(* PLC project Generated.project, CODESYS CODESYS V3.5 SP19 Patch 1 *)
(* stored: creationDateTime 2026-07-27T13:56:34.388274, modificationDateTime 2026-07-27T13:56:34.388274 *)

TYPE ST_Chain_Winch_Demandes : STRUCT
  Idx201_JoyRawPhysical_ANA : INT;  (* [pts] Bruts convertisseur (-2048 à +2048) *)
  Idx202_JoyScaledPhysical_Pct : REAL;  (* [%] Consigne Joystick (-100% à +100%) *)
  Idx203_HmiManualCmd_BtnUp : BOOL;  (* 1 = Appui Bouton Montée IHM | 0 = Relâché *)
  Idx204_HmiManualCmd_BtnDown : BOOL;  (* 1 = Appui Bouton Descente IHM | 0 = Relâché *)
  Idx205_CycleAutoCmd_Pct : REAL;  (* [%] Consigne auto envoyée par le Cycle *)
  Idx206_ModeActive : E_Mode;  (* Mode courant (MANU_N1, AUTO_N1, MAINT_N2...) *)
  Idx207_BypassOperatorComm : BOOL;  (* 0 = Comm Normale OK | 1 = Bypass Réseau Actif ⚠️ *)
  Idx208_ArbitratedSpeed_Pct : REAL;  (* [%] Consigne finale retenue après arbitrage *)
  Idx209_ArbitratedDirection : INT;  (* +1 = Montée | 0 = Neutre | -1 = Descente *)
END_STRUCT;
END_TYPE

(* values of E_Mode: DISABLE: Mode Désactivé / Veille de sécurité (sorties bloquées); MAINT_N1: Manuel Niveau 1 : Pilotage unitaire avec toutes sécurités actives; MAINT_N2: Manuel Niveau 2 : Pilotage dégradé (droits étendus + bypasses autorisés); SEMI_AUTO: Mode Semi-Automatique (séquenceur automatique) *)

{attribute 'qualified_only'}
{attribute 'strict'}
TYPE E_Mode : (DISABLE := 0, MAINT_N1 := 1, MAINT_N2 := 2, SEMI_AUTO := 3);
END_TYPE
